(*********************************** G.D S.p.A. - Technical Department ***********************************
============= PROGRAM INFO ============
FOLDER:             TBD
MACHINES INVOLVED:  TBD 

============= DESCRIPTION =============
csp machine declaration

============= REVISIONS ===============
Date		Version	 	Author      	Description             
----------	-------		------------  	--------------------------------------------
2019/04/05 	0000.00	 	M.Grasso		Creation of the PRG

**********************************************************************************************************)
(*$R process_ref := prc; $*)
PROGRAM csp_transfer_infeed_waterfall
VAR
	
	prc:									process;
	prc_path:								STRING;
	
	
	waterfall_conveyor_running:				BOOL;
	disable_req:							BOOL;
	
END_VAR

_read_var_input();

_object_manager();

IF NOT objects_running()
THEN
	RETURN;	
END_IF

_read_process_image();

_mode_manager();

CASE process_get_mode(prc) OF
	MODE_ABSENT,
	MODE_INACTIVE:
		RETURN;
	MODE_TEST:
		_handle_process_test();
END_CASE


_set_runtime_properties();

(********************************* BODY *********************************)
(************************************************************************)

waterfall_conveyor_running := axis_is_moving(csp_transfer_infeed_waterfall_belt.axis);

disable_req := NOT
				(
					(
					csp_transfer_infeed.run_infeed_belts
					)
					AND
					process_is_ready(prc)
					AND
					process_subtree_is_ready(prc)
				);

_handle_messages();

_write_output();

ACTION _handle_messages:
;
END_ACTION

ACTION _handle_process_test:
;
END_ACTION

ACTION _mode_manager:
IF process_mode_req_is_pending(prc)
THEN
    process_apply_mode_req_first_step(prc);
    CASE process_get_mode(prc) OF
        MODE_TO_ABSENT:
			;
        MODE_TO_INACTIVE:
			;
        MODE_TO_TEST:
			;
        MODE_TO_OPERATIONAL:
			;
    END_CASE
    process_apply_mode_req_second_step(prc);
END_IF
END_ACTION

ACTION _object_manager:
IF objects_initialization()
THEN
	sub_process_init(
		object_name					:= 'csp_transfer_infeed_waterfall.prc', 
		process						:= csp_transfer_infeed.prc, 
		CONVERSION_this				:= prc);
		
	prc_path 						:= process_get_path(prc);
	
END_IF

IF objects_running()
THEN
	process_cycle(prc);

END_IF
END_ACTION

ACTION _read_process_image:
;
END_ACTION

ACTION _read_var_input:
;
END_ACTION

ACTION _set_runtime_properties:
;
END_ACTION

ACTION _write_output:
;
END_ACTION

END_PROGRAM

(* stored: Version 1.1.0.1, ProductVersion 3.1.4024.3
   POU csp_transfer_infeed_waterfall: Id {41c0ead2-71c6-4d94-8fd5-0536c646177e}, SpecialFunc None
   Action _handle_messages: Id {a9d3aee3-c580-4d65-b4d5-20b5fdcd9182}
   Action _handle_process_test: Id {ad98a837-ae68-4a6e-adea-91f8ea2aa17b}
   Action _mode_manager: Id {b8c0c636-5969-4347-a24a-8bbea1f148e5}
   Action _object_manager: Id {3587963b-0157-4328-9f94-f71bd522b512}
   Action _read_process_image: Id {75e05b5c-2c92-4df0-8a3e-14b49f5d0cbf}
   Action _read_var_input: Id {8de5a476-458b-46cd-93c3-79aa26ebc4f4}
   Action _set_runtime_properties: Id {d42ffba5-b175-425c-9d76-b527dc3d4f90}
   Action _write_output: Id {f7644f50-ad4a-4250-b031-1e2acf1b5e94} *)
